(* PLC project Proj1, GeneratedByPython TwinCAT PLC Control 3.5.x *)
(* stored: creationDateTime 2026-01-21T07:07:40, modificationDateTime 2026-01-21T07:07:40 *)

FUNCTION_BLOCK FB_GeneratedJob_01
  VAR
    eState : INT;
    bFinished : BOOL;
    nCounter : INT;
    fResult : LREAL;
  END_VAR

// Haupt-Body des FBs - ruft State Machine Logik auf
// Hier könnte auch zyklischer Code stehen

METHOD JobStart : BOOL
// Methode: JobStart
eState := 1;
bFinished := FALSE;
nCounter := 0;
fResult := 0.0;
JobStart := TRUE;
END_METHOD

METHOD Abort : BOOL
// Methode: Abort
eState := 4;
bFinished := FALSE;
Abort := TRUE;
END_METHOD

METHOD CheckState : INT
// Methode: CheckState (Zyklisch aufgerufen)
CASE eState OF
    0:
        ; // Warten auf Start

    1:
        // --- HIER KOMMT DEIN GENERIERTER CODE REIN ---
        
// Dies ist der Code, den wir vorher generiert haben
nCounter := nCounter + 1;
fResult := SQRT(REAL_TO_LREAL(nCounter));

IF nCounter > 100 THEN
    bFinished := TRUE;
END_IF

        // ---------------------------------------------

        IF bFinished THEN
            eState := 2;
        END_IF

    2:
        ; // Fertig

    3:
        ; // Fehlerbehandlung

    4:
        eState := 0; // Reset nach Abort
END_CASE
CheckState := eState;
END_METHOD
END_FUNCTION_BLOCK
